SUBAPPLICATION Uebung_033_sub (* LED Strip Blinkende LED *)
  (* Standard: 61499-2; Description: Copyright (c) 2023 Meisterschulen am Ostbahnhof This program and the accompanying materials are made available under the terms of the Eclipse Public License 2.0 which is available at https://www.eclipse.org/legal/epl-2.0/ SPDX-License-Identifier: EPL-2.0 *)
  (* Version 1.0, 2023-10-23, Franz Höpfinger, Meisterschulen am Ostbahnhof *)
  IMPORT logiBUS::io::DI::logiBUS_DI_S;
  IMPORT logiBUS::io::DO_LED::LED_COLOURS;
  IMPORT logiBUS::io::DO_LED::LED_FREQ;
  IMPORT logiBUS::io::DI::logiBUS_DI::Invalid;
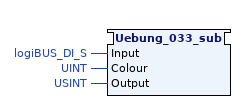
  VAR_INPUT
    Input : logiBUS::io::DI::logiBUS_DI_S := Invalid; (* Identify the Input Input_I1..I8 *)
    Colour : UINT := LED_COLOURS::LED_GREEN; (* This identify the Colour. *)
    Output : USINT; (* Identify the Output Number of Strip *)
  END_VAR
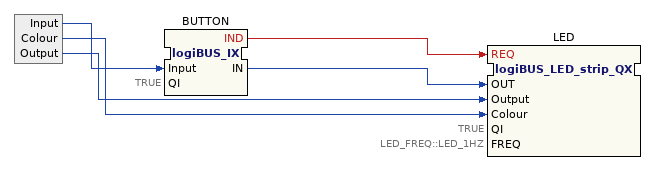
  FBS
    LED : logiBUS::io::DO_LED::logiBUS_LED_strip_QX(QI := TRUE, FREQ := LED_FREQ::LED_1HZ);
    BUTTON : logiBUS::io::DI::logiBUS_IX(QI := TRUE);
  END_FBS
  EVENT_CONNECTIONS
    BUTTON.IND TO LED.REQ;
  END_CONNECTIONS
  DATA_CONNECTIONS
    BUTTON.IN TO LED.OUT;
    Input TO BUTTON.Input;
    Output TO LED.Output;
    Colour TO LED.Colour;
  END_CONNECTIONS
END_SUBAPPLICATION
